// TIA Portal V20 export
FUNCTION_BLOCK "FB_FixtureV_Init"   // FB77, SCL
{ S7_Optimized_Access := 'TRUE' }
// stored: AutoNumber false, MemoryReserve 100, SetENOAutomatically false
   VAR_INPUT
      iStartSeqCond : Bool;   // Start Sequence Conditions
      iJobReq : Bool;   // Job Request - From Main
      iAxisV_FixtSafePos : Bool;
      iAxisV_FixtSafePosSetPoint : LReal;
      iAxisV_Moving : Bool;   // Shuttle is moving
      iAxisV_InPos : Bool;
      iPLC_DateAndTime : DTL;
      iStepPause : Bool;
   END_VAR
   VAR_OUTPUT
      oAxisV_StartReq : Bool;
      oAxisV_PosSetPoint : Real;
   END_VAR
   VAR
      sCurrent_Step_NB : Int;   // Active Step Number
      sCheck_Step_Condition : Bool;
      sOneStepForward : Bool;
      sRTOneStepForward : R_TRIG;
      sOneStepMode { S7_SetPoint := 'True'} : Bool;
      sStepForward : Bool;
      sInterface : "UDT_SequenceInterface";
      sAxisV_StartReq : Bool;
      sAxisV_PosSetPoint : Real;
      sHistory : Struct
         Activation : Bool;
         Steps : Array[0..99] of Int;
         Date_Time : Array[0..99] of DTL;
      END_STRUCT;
      StepText : "FB_GetTextErrorCode";
   END_VAR
   VAR_TEMP
      tIndex : Int;   // Index
   END_VAR
   VAR CONSTANT
      S00_INIT : Int := 0;
      S10_CHECK_FIXTURE_RELEASE_OPTION : Int := 10;
      S20_AXIS_V_TO_FIXTURE_SAFE_POS_START_REQ : Int := 20;
      S30_AXIS_V_TO_FIXTURE_SAFE_POS_REACHED : Int := 30;
      S95_JOB_DONE : Int := 95;
   END_VAR
   // StepText.sCode_error[0].ErrorCode := 0;
   // StepText.sCode_error[1].ErrorCode := 10;
   // StepText.sCode_error[2].ErrorCode := 20;
   // StepText.sCode_error[3].ErrorCode := 30;
   // StepText.sCode_error[4].ErrorCode := 40;
   // StepText.sCode_error[5].ErrorCode := 50;
   // StepText.sCode_error[6].ErrorCode := 60;
   // StepText.sCode_error[7].ErrorCode := 70;
   // StepText.sCode_error[8].ErrorCode := 80;
   // StepText.sCode_error[9].ErrorCode := 90;
   // StepText.sCode_error[10].ErrorCode := 95;
BEGIN
   REGION Description header 
       //==================================================================================
       // POSALUX Swiss SA / (C) Copyright 2026
       //----------------------------------------------------------------------------------
       // Title: FB_FixtureV_Init
       // Comment/Function: 
       // Author: Fabien WALDT
       // Engineering: TIA Portal v20
       //----------------------------------------------------------------------------------
       // Change log table:
       // Version  | Date     | Expert in charge | Changes applied
       // ---------|----------|------------------|-----------------------------------------
       // 00.00.01 | 20260220 | WFA              | First released version
       // =================================================================================
   END_REGION

   REGION Define condition to start
       IF #iStartSeqCond THEN
           #sInterface.SequenceReleased := TRUE;
       ELSE
           // Standard sequencer controls
           #sInterface.SequenceReleased := FALSE;
           #sCurrent_Step_NB := #S00_INIT;
           #sInterface.SequenceRun := FALSE;
           #sInterface.JobDone := FALSE;
           #sCheck_Step_Condition := FALSE;

           // Dedicated sequencer controls
           #sAxisV_StartReq := FALSE;
           #sAxisV_PosSetPoint := 0.0;

           // Add specifics controls 
       END_IF;

       // Reset interface error
       IF #sInterface.Reset THEN
           #sInterface.Error := FALSE;
       END_IF;

       // Reset start when axis in position
       IF #iAxisV_InPos THEN
           #sAxisV_StartReq := FALSE;
       END_IF;

       // One step forward
       #sRTOneStepForward.CLK := #sOneStepForward;
       #sRTOneStepForward();
       #sStepForward := (NOT #sOneStepMode OR (#sOneStepMode AND #sRTOneStepForward.Q)) AND NOT #iStepPause;
       #sOneStepForward := FALSE;

       // Action only true in dedicated steps

       // Step Timer

   END_REGION

   REGION Sequence Function
       CASE #sCurrent_Step_NB OF
           #S00_INIT:
               REGION S00 INIT
                   #sCheck_Step_Condition := TRUE;
               END_REGION
           #S10_CHECK_FIXTURE_RELEASE_OPTION:
               REGION S10_CHECK_FIXTURE_RELEASE_OPTION
                   #sCheck_Step_Condition := TRUE;
               END_REGION
           #S20_AXIS_V_TO_FIXTURE_SAFE_POS_START_REQ:
               REGION S20_AXIS_V_TO_FIXTURE_SAFE_POS_START_REQ
                   #sAxisV_StartReq := NOT #iAxisV_FixtSafePos;
                   #sAxisV_PosSetPoint := LREAL_TO_REAL(#iAxisV_FixtSafePosSetPoint);
                   #sCheck_Step_Condition := TRUE;
               END_REGION
           #S30_AXIS_V_TO_FIXTURE_SAFE_POS_REACHED:
               REGION S30_AXIS_V_TO_FIXTURE_SAFE_POS_REACHED
                   #sCheck_Step_Condition := TRUE;
               END_REGION
           #S95_JOB_DONE:
               REGION S95_JOB_DONE
                   #sInterface.JobDone := TRUE;
                   #sCheck_Step_Condition := TRUE;
               END_REGION
           ELSE:
               #sInterface.Error := TRUE;
       END_CASE;
   END_REGION

   REGION Sequence Next Step Condition
       IF #sCheck_Step_Condition THEN
           CASE #sCurrent_Step_NB OF
               #S00_INIT:
                   REGION S00_INIT
                       IF #sInterface.SequenceReleased AND #iJobReq THEN
                           #sCurrent_Step_NB := #S10_CHECK_FIXTURE_RELEASE_OPTION;
                           #sInterface.SequenceRun := TRUE;
                           #sCheck_Step_Condition := FALSE;
                       ELSE
                           #sInterface.SequenceRun := FALSE;
                       END_IF;
                   END_REGION
               #S10_CHECK_FIXTURE_RELEASE_OPTION:
                   REGION S10_CHECK_FIXTURE_RELEASE_OPTION
                       IF #sInterface.SequenceReleased AND #sStepForward AND NOT "DB_LoaderOptions".Fixture.V_InitDisabled THEN
                           #sCurrent_Step_NB := #S20_AXIS_V_TO_FIXTURE_SAFE_POS_START_REQ;
                           #sCheck_Step_Condition := FALSE;
                       ELSIF #sInterface.SequenceReleased AND #sStepForward AND "DB_LoaderOptions".Fixture.V_InitDisabled THEN
                           #sCurrent_Step_NB := #S95_JOB_DONE;
                           #sCheck_Step_Condition := FALSE;
                       END_IF;
                   END_REGION
               #S20_AXIS_V_TO_FIXTURE_SAFE_POS_START_REQ:
                   REGION S20_AXIS_V_TO_FIXTURE_SAFE_POS_START_REQ
                       IF #sInterface.SequenceReleased AND #sStepForward AND (#iAxisV_Moving OR #iAxisV_FixtSafePos) THEN
                           #sCurrent_Step_NB := #S30_AXIS_V_TO_FIXTURE_SAFE_POS_REACHED;
                           #sCheck_Step_Condition := FALSE;
                       END_IF;
                   END_REGION
               #S30_AXIS_V_TO_FIXTURE_SAFE_POS_REACHED:
                   REGION S30_AXIS_V_TO_FIXTURE_SAFE_POS_REACHED
                       IF #sInterface.SequenceReleased AND #sStepForward AND NOT #sAxisV_StartReq AND #iAxisV_FixtSafePos THEN
                           #sCurrent_Step_NB := #S95_JOB_DONE;
                           #sCheck_Step_Condition := FALSE;
                       END_IF;
                   END_REGION
               #S95_JOB_DONE:
                   REGION S95_JOB_DONE
                       IF NOT #iJobReq THEN
                           #sCurrent_Step_NB := #S00_INIT;
                           #sCheck_Step_Condition := FALSE;
                           #sInterface.JobDone := FALSE;
                       END_IF;
                   END_REGION
               ELSE
                   #sInterface.Error := TRUE;
           END_CASE;
       END_IF;
   END_REGION

   REGION Outputs Update
       #oAxisV_StartReq := #sAxisV_StartReq;
       #oAxisV_PosSetPoint := #sAxisV_PosSetPoint;
   END_REGION

   REGION Steps - Date and Time History
       IF #sHistory.Activation THEN
           IF #sHistory.Steps[0] <> #sCurrent_Step_NB THEN
               FOR #tIndex := 98 TO 0 BY -1 DO
                   #sHistory.Steps[#tIndex + 1] := #sHistory.Steps[#tIndex];
                   #sHistory.Date_Time[#tIndex + 1] := #sHistory.Date_Time[#tIndex];
               END_FOR;
               #sHistory.Steps[0] := #sCurrent_Step_NB;
               #sHistory.Date_Time[0] := #iPLC_DateAndTime;
           END_IF;
       END_IF;
   END_REGION

   REGION Steps Text
       #StepText(iErrorCode := #sCurrent_Step_NB,
                 oErrorText => #StepText.oErrorText);
   END_REGION
END_FUNCTION_BLOCK
